TYPE FB_Interpolation_State :
(
	UNDEFINIERT := 0,
	STAND_BY,
	ENABLE,
	FAHRE_ABSOLUT,
	HAND_Y_POS,
	HAND_Y_NEG,
	HAND_X_POS,
	HAND_X_NEG,
	ERROR_HANDLER
);
END_TYPE

(* stored: Version 1.1.0.1, ProductVersion 3.1.4018.5
   DUT FB_Interpolation_State: Id {1c1110b6-4085-4778-8bc9-e14be883e8f4} *)
